FUNCTION_BLOCK CU020ManualTask EXTENDS TcoTaskedService IMPLEMENTS ICUTask
VAR
END_VAR

Run();

(*~
	<docu>
		<summary>
			Main method of the sequener. Custom code needs to be placed here. The sequencer is executed by call of **Instance.Run()** method.
			This method is abstract, and it must be overridden in derived block.
		</summary>
	</docu>
~*)
METHOD PROTECTED Main : BOOL
Messenger.Notify('Running manual mode');
Station.Components.Group1.horizontalCylinder.Service();
END_METHOD

METHOD PROTECTED OnStart
Station.AutomatTask.Restore();
Station.GroundTask.Restore();
Station.GroundTask.CancelGround();
END_METHOD

PROPERTY Station : REFERENCE TO CU020
GET
VAR
    _station : POINTER TO CU020;
END_VAR
IF __QUERYPOINTER(Parent, _station) THEN // Check if _Parent is Station001
    Station REF= _station^;              // If the check is successful dereference a pointer. simlar to THIS^ or SUPER^
END_IF
END_GET
END_PROPERTY

END_FUNCTION_BLOCK

(* stored: Version 1.1.0.1
   POU CU020ManualTask: Id {1af38a75-db48-4ffa-915c-7a7d705d39bc}, SpecialFunc None
   Method Main: Id {91569f3f-a7a0-41fa-9d52-adc26d855830}
   Method OnStart: Id {7e096d7f-2863-4523-8cef-604315d91c6c}
   Property Station: Id {4e553048-1c91-4ee4-a72c-26f122cabf45}
   Get Get: Id {67857616-7a80-4485-be51-2302cfd8df6b} *)
